// TIA Portal V19 export
VAR_GLOBAL   // PLC tag table "Default tag table"
   Axis_1_Drive_IN AT %I68.0 : "PD_TEL3_IN";
   Axis_1_Drive_OUT AT %Q82.0 : "PD_TEL3_OUT";
   "Axis_1_Homing switch" AT %I0.3 : Bool;
   firstscan AT %M10.0 : Bool;
   "Homing procedure" AT %M11.0 : Bool;
   Home_Done_Vertical AT %M11.1 : Bool;
   Tag_1 AT %I2.0 : Bool;
   Tag_2 AT %M20.0 : Bool;
   ServoONHorizont AT %Q0.7 : Bool;
   home_horizontal AT %Q0.4 : Bool;
   Home_done_horizontal AT %M12.0 : Bool;
   HomeComplete AT %I8.0 : Bool;
   Tag_3 AT %I1.3 : Bool;
   Servo_fault AT %I1.4 : Bool;
   Servo_Alarm AT %I1.5 : Bool;
   Tag_4 AT %M100.0 : Bool;
   System_Byte AT %MB8001 : Byte;
   "FirstScan(1)" AT %M1.0 : Bool;
   DiagStatusUpdate AT %M8001.1 : Bool;
   AlwaysTRUE AT %M8001.2 : Bool;
   AlwaysFALSE AT %M8001.3 : Bool;
   Clock_Byte AT %MB8000 : Byte;
   Clock_10Hz AT %M8000.0 : Bool;
   Clock_5Hz AT %M8000.1 : Bool;
   "Clock_2.5Hz" AT %M8000.2 : Bool;
   Clock_2Hz AT %M8000.3 : Bool;
   "Clock_1.25Hz" AT %M8000.4 : Bool;
   Clock_1Hz AT %M8000.5 : Bool;
   "Clock_0.625Hz" AT %M8000.6 : Bool;
   "Clock_0.5Hz" AT %M8000.7 : Bool;
   Tag_5 AT %M100.1 : Bool;
   Reset_HorizontDrive AT %Q0.6 : Bool;
   "hent 8cm" AT %M1000.0 : Bool;
   Binær_hent_8cm AT %M50.0 : Bool;
   Stepdata_1_U AT %Q0.1 : Bool;
   Stepdata_2_U AT %Q0.2 : Bool;
   Stepdata_3_U AT %Q0.3 : Bool;
   Stepdata_1_Conf AT %I0.6 : Bool;
   Stepdata_2_Conf AT %I0.7 : Bool;
   Stepdata_3_Conf AT %I1.0 : Bool;
   Drive_Servo AT %Q0.5 : Bool;
   lever_8cm AT %M1000.1 : Bool;
   "binær _lever_8cm" AT %M50.1 : Bool;
   "Sett sylinder C7" AT %M50.7 : Bool;
   "Sylinder C7" AT %Q0.0 : Bool;
   Tag_8 AT %M50.2 : Bool;
   Hent_16cm AT %M50.4 : Bool;
   Binær_Hent_16cm AT %M50.5 : Bool;
   Lever_16cm AT %M50.6 : Bool;
   binær_lever_16cm AT %M51.0 : Bool;
END_VAR
